# EPICS substitutions: EUROTHRM/EUROTHRM-IOC-01App/Db/devEurothrmA04.substitutions
# Note: this file is generated by generate_substitutions.py
file devEurothrm.template {
pattern { P, GAD, LAD, MODBUS_PV, MODBUS_SP, MODBUS_P, MODBUS_I, MODBUS_D, MODBUS_HS, MODBUS_LS, MODBUS_AT, MODBUS_HO, MODBUS_OP }
{ "\$(P)", "0", "4", "3073", "3074", "3078", "3080", "3081", "3183", "3184", "3342", "3102", "3075" }
}
